FUNCTION_BLOCK MaterialHolder
VAR_IN_OUT
	slots : ARRAY[*] OF STRING;
	occupied : ARRAY[*] OF BOOL;
	
	hmiTable : ARRAY[*] OF MaterialSlot;
END_VAR
VAR
	numSlots : INT;
END_VAR

(*
by default:
	hmiTable contains the true data, including IO mapped to hardware
	slots and occupied cyclically copy data from hmiTable

if hmiTable is NULL (not passed in), then slots and occupied will store the true data
	
the program will access data using slots/occupied via methods
when the data is changed, data is copied from slots/occupied to hmiTable

this ensures that the methods update the HMI, and the HMI updates the data
*)


IF hmiTable <> 0 AND_THEN (slots <> 0  AND occupied <> 0) THEN
	writeArrays();
END_IF

numSlots := TO_INT(UPPER_BOUND(slots, 1) - LOWER_BOUND(slots, 1) + 1);

METHOD clear : BOOL
VAR_INPUT
END_VAR
MEMSET(ADR(slots), 0, SIZEOF(slots));
END_METHOD

METHOD findSlot : BOOL
VAR_INPUT
	materialID : STRING;
END_VAR
VAR_OUTPUT
	atPosition : INT := -1;
END_VAR
VAR
	i : INT;
END_VAR
(*
IF materialID = '' THEN
	RETURN;
END_IF
*)
FOR i:=1 TO GVL.maxQueue BY 1 DO
	IF slots[i] = materialID THEN
		atPosition := i;
		findSlot := TRUE;
		RETURN;
	END_IF
END_FOR
END_METHOD

METHOD getSlot : STRING
VAR_INPUT
	i : DINT;
END_VAR
VAR_OUTPUT
	errorBounds : BOOL;
END_VAR
errorBounds := i < LOWER_BOUND(slots, 1) OR i > UPPER_BOUND(slots, 1);

IF errorBounds THEN
	RETURN;
END_IF

getSlot := slots[i];
END_METHOD

METHOD getSlotsAsArray : POINTER TO STRING
getSlotsAsArray := ADR(slots);
END_METHOD

METHOD isOccupied : BOOL
VAR_INPUT
	i : DINT;
END_VAR
VAR_OUTPUT
	errorBounds : BOOL;
END_VAR
errorBounds := i < LOWER_BOUND(slots, 1) OR i > UPPER_BOUND(slots, 1);

IF errorBounds THEN
	RETURN;
END_IF

isOccupied := occupied[i];
END_METHOD

METHOD setSlot : BOOL
VAR_INPUT
	i : INT;
	material : STRING;
END_VAR
VAR_OUTPUT
	error : BOOL;
END_VAR
IF i < LOWER_BOUND(slots, 1) OR i > UPPER_BOUND(slots, 1) THEN
	error := TRUE;
	RETURN;
END_IF

slots[i] := material;

IF hmiTable <> 0 THEN
	writeHmiTable();
END_IF
END_METHOD

METHOD PROTECTED writeArrays : BOOL
VAR
	i : DINT;
END_VAR
FOR i:=LOWER_BOUND(hmiTable, 1) TO UPPER_BOUND(hmiTable, 1) BY 1 DO
	slots[i] := hmiTable[i].material;
	occupied[i] := hmiTable[i].occupied;
END_FOR
END_METHOD

METHOD PROTECTED writeHmiTable : BOOL
VAR
	i : DINT;
END_VAR
FOR i:=LOWER_BOUND(hmiTable, 1) TO UPPER_BOUND(hmiTable, 1) BY 1 DO
	hmiTable[i].material := slots[i];
	hmiTable[i].occupied := occupied[i];
END_FOR
END_METHOD

END_FUNCTION_BLOCK

(* stored: Version 1.1.0.1, ProductVersion 3.1.4024.11
   POU MaterialHolder: Id {b8766d7a-1d6a-4377-9cc8-53e16c54b972}, SpecialFunc None
   Folder HMI: Id {e0175151-2858-4df9-807d-10c6bd8b5349}
   Method clear: Id {0079e54a-4897-43fe-babe-0b16afa40b6d}
   Method findSlot: Id {584be88a-e8b0-4046-8e86-717c358b8f08}
   Method getSlot: Id {de92b67f-dd7e-4c53-9c6e-8ccbe92049e8}
   Method getSlotsAsArray: Id {dff81b33-35f2-4bb2-b5f5-baf2f77d8ad6}
   Method isOccupied: Id {e248ac69-fb6d-46e9-aac8-29ec13f4c904}
   Method setSlot: Id {b2a4e65d-50f3-4f46-a49d-166b867372cc}
   Method writeArrays: Id {a5628a64-2b8c-4bd1-880c-5e15b3abea8a}
   Method writeHmiTable: Id {f1391623-2367-48f0-8486-56e290217047} *)
